// TIA Portal V17 export
// export: Created 2023-02-14T02:49:13.2032669Z, ExportSetting WithDefaults, DisplayName Totally Integrated Automation Portal, DisplayVersion V17, DisplayName TIA Portal Openness, DisplayVersion V17, DisplayName TIA Portal Teamcenter Gateway, DisplayVersion V17, DisplayName TIA Portal Version Control Interface, DisplayVersion V17, DisplayName SINAMICS Startdrive Advanced, DisplayVersion V17, DisplayName SINAMICS Startdrive G130, G150, S120, S150, SINAMICS MV, S210, DisplayVersion V17, DisplayName SINAMICS Startdrive G110M, G120, G120C, G120D, G120P, G115D, DisplayVersion V17, DisplayName STEP 7 Professional, DisplayVersion V17, DisplayName STEP 7 Safety, DisplayVersion V17, DisplayName WinCC Professional, DisplayVersion V17
DATA_BLOCK "Mix_to_CIP"   // DB221
{ S7_Optimized_Access := 'FALSE' }
VERSION : 0.1
// stored: AutoNumber false, DBAccessibleFromOPCUA true, DBAccessibleFromWebserver true, IsOnlyStoredInLoadMemory false, IsWriteProtectedInAS false
   VAR
      HeartBeat : Bool := TRUE;
      CIP_Request : Struct
         Header : Struct
            Header_CIP_Request : Bool;
         END_STRUCT;
         "Chili Awetan" : Struct
            "T-02.00_CIP_Request" : Bool;
            "T-03.00_CIP_Request" : Bool;
            "T-04.00_CIP_Request" : Bool;
         END_STRUCT;
         Tomato : Struct
            "T-05.00_CIP_Request" : Bool;
         END_STRUCT;
         ChiliFresh : Struct
            "T-06.00_CIP_Request" : Bool;
            "T-07.00_CIP_Request" : Bool;
            "T-08.00_CIP_Request" : Bool;
         END_STRUCT;
         Garlic : Struct
            "T-09.00_CIP_Request" : Bool;
         END_STRUCT;
         Vinegar : Struct
            "T-10.00_CIP_Request" : Bool;
         END_STRUCT;
         Homomixer : Struct
            "T-12.00_CIP_Tank_Request" : Bool;
            "T-12.00_CIP_LineToBlend_Request" : Bool;
            "T-13.00_CIP_Tank_Request" : Bool;
            "T-13.00_CIP_LineToBlend_Request" : Bool;
            "T-14.00_CIP_Tank_Request" : Bool;
            "T-14.00_CIP_LineToBlend_Request" : Bool;
         END_STRUCT;
         "Blending Cluster 1" : Struct
            "T-20.00_CIP_Request" : Bool;
            "T-21.00_CIP_Request" : Bool;
            "T-30.00_CIP_Request" : Bool;
            Blending_Cluster1_LineProduct_Request : Bool;
            Free_CIP_Req_1 : Bool;
            Free_CIP_Req_2 : Bool;
         END_STRUCT;
         "Blending Cluster 2" : Struct
            "T-31.00_CIP_Request" : Bool;
            "T-40.00_CIP_Request" : Bool;
            "T-41.00_CIP_Request" : Bool;
            Blending_Cluster2_LineProduct_Request : Bool;
            Free_CIP_Req_1 : Bool;
            Free_CIP_Req_2 : Bool;
         END_STRUCT;
         "Rework Cluster 1" : Struct
            "T-22.00_CIP_Request" : Bool;
         END_STRUCT;
         "Rework Cluster 2" : Struct
            "T-32.00_CIP_Request" : Bool;
         END_STRUCT;
         "Buffer Cluster 1" : Struct
            "T-61.00_CIP_Request" : Bool;
            "T-62.00_CIP_Request" : Bool;
            "T61&T62_CIP_LineToPasteur_Request" : Bool;
            "T-63.00_CIP_Request" : Bool;
            "T-64.00_CIP_Request" : Bool;
            "T63&T64_CIP_LineToPasteur_Request" : Bool;
         END_STRUCT;
         "Buffer Cluster 2" : Struct
            "T-65.00_CIP_Request" : Bool;
            "T-66.00_CIP_Request" : Bool;
            "T65&T66_CIP_LineToPasteur_Request" : Bool;
            "T-67.00_CIP_Request" : Bool;
            "T-68.00_CIP_Request" : Bool;
            "T67&T68_CIP_LineToPasteur_Request" : Bool;
         END_STRUCT;
         "Storage THE 4" : Struct
            "T-23.00_CIP_Tank_Request" : Bool;
            "T-23.00_CIP_Line_Request" : Bool;
            "T-24.00_CIP_Tank_Request" : Bool;
            "T-24.00_CIP_Line_Request" : Bool;
            THE4_LineProduct_CIP_Request : Bool;
         END_STRUCT;
         "Storage THE 5" : Struct
            "T-33.00_CIP_Tank_Request" : Bool;
            "T-34.00_CIP_Tank_Request" : Bool;
            "T33&T34_CIP_Line_Request" : Bool;
            "T-35.00_CIP_Tank_Request" : Bool;
            "T-35.00_CIP_Line_Request" : Bool;
            THE5_LineProduct_CIP_Request : Bool;
         END_STRUCT;
         "T-79.00_CIP_Tank_Request" : Bool;
         "T-79.00_CIP_Line_Request" : Bool;
         "T-81.00_CIP_Request" : Bool;
         "T-84.00_CIP_Request" : Bool;
         "T-85.00_CIP_Request" : Bool;
         Free_CIP_Req_6 : Bool;
         Free_CIP_Req_7 : Bool;
         Free_CIP_Req_8 : Bool;
         Free_CIP_Req_9 : Bool;
         Free_CIP_Req_10 : Bool;
         Free_CIP_Req_11 : Bool;
         Free_CIP_Req_12 : Bool;
         Free_CIP_Req_13 : Bool;
         Free_CIP_Req_14 : Bool;
         Free_CIP_Req_15 : Bool;
         Free_CIP_Req_16 : Bool;
         Osa_CIP_Req : Bool;
         Free_CIP_Req_18 : Bool;
         Free_CIP_Req_19 : Bool;
         Free_CIP_Req_20 : Bool;
         Free_CIP_Req_21 : Bool;
         Free_CIP_Req_22 : Bool;
         Free_CIP_Req_23 : Bool;
         Free_CIP_Req_24 : Bool;
      END_STRUCT;
      CIP_Line_OK : Struct
         Header : Struct
            Header_CIP_LineOK : Bool;
         END_STRUCT;
         "Chili Awetan" : Struct
            "T-02.00_CIP_LineOK" : Bool;
            "T-03.00_CIP_LineOK" : Bool;
            "T-04.00_CIP_LineOK" : Bool;
         END_STRUCT;
         Tomato : Struct
            "T-05.00_CIP_LineOK" : Bool;
         END_STRUCT;
         ChiliFresh : Struct
            "T-06.00_CIP_LineOK" : Bool;
            "T-07.00_CIP_LineOK" : Bool;
            "T-08.00_CIP_LineOK" : Bool;
         END_STRUCT;
         Garlic : Struct
            "T-09.00_CIP_LineOK" : Bool;
         END_STRUCT;
         Vinegar : Struct
            "T-10.00_CIP_LineOK" : Bool;
         END_STRUCT;
         Homomixer : Struct
            "T-12.00_CIP_LineOK" : Bool;
            "T-13.00_CIP_LineOK" : Bool;
            "T-14.00_CIP_LineOK" : Bool;
         END_STRUCT;
         "Blending Cluster 1" : Struct
            "T-20.00_CIP_LineOK" : Bool;
            "T-21.00_CIP_LineOK" : Bool;
            "T-30.00_CIP_LineOK" : Bool;
            Blending_Cluster1_LineProduct_LineOK : Bool;
            Free_CIP_LineOK_1 : Bool;
            Free_CIP_LineOK_2 : Bool;
         END_STRUCT;
         "Blending Cluster 2" : Struct
            "T-31.00_CIP_LineOK" : Bool;
            "T-40.00_CIP_LineOK" : Bool;
            "T-41.00_CIP_LineOK" : Bool;
            Blending_Cluster2_LineProduct_LineOK : Bool;
            Free_CIP_LineOK_1 : Bool;
            Free_CIP_LineOK_2 : Bool;
         END_STRUCT;
         "Rework Cluster 1" : Struct
            "T-22.00_CIP_LineOK" : Bool;
         END_STRUCT;
         "Rework Cluster 2" : Struct
            "T-32.00_CIP_LineOK" : Bool;
         END_STRUCT;
         "Buffer Cluster 1" : Struct
            "T-61.00_CIP_LineOK" : Bool;
            "T-62.00_CIP_LineOK" : Bool;
            "T61&T62_CIP_LineToPasteur_LineOK" : Bool;
            "T-63.00_CIP_LineOK" : Bool;
            "T-64.00_CIP_LineOK" : Bool;
            "T63&T64_CIP_LineToPasteur_LineOK" : Bool;
         END_STRUCT;
         "Buffer Cluster 2" : Struct
            "T-65.00_CIP_LineOK" : Bool;
            "T-66.00_CIP_LineOK" : Bool;
            "T65&T66_CIP_LineToPasteur_LineOK" : Bool;
            "T-67.00_CIP_LineOK" : Bool;
            "T-68.00_CIP_LineOK" : Bool;
            "T67&T68_CIP_LineToPasteur_LineOK" : Bool;
         END_STRUCT;
         "Storage THE 4" : Struct
            "T-23.00_CIP_LineOK" : Bool;
            "T-24.00_CIP_LineOK" : Bool;
            THE4_LineProduct_CIP_LineOK : Bool;
         END_STRUCT;
         "Storage THE 5" : Struct
            "T-33.00_CIP_Tank_LineOK" : Bool;
            "T-34.00_CIP_Tank_LineOK" : Bool;
            "T33&T34_CIP_Line_LineOK" : Bool;
            "T-35.00_CIP_Tank_LineOK" : Bool;
            THE5_LineProduct_CIP_LineOK : Bool;
         END_STRUCT;
         "T-79.00_CIP_LineOK" : Bool;
         "T-81.00_CIP_LineOK" : Bool;
         "T-84.00_CIP_LineOK" : Bool;
         "T-85.00_CIP_LineOK" : Bool;
         Free_CIP_LineOK_5 : Bool;
         Free_CIP_LineOK_6 : Bool;
         Free_CIP_LineOK_7 : Bool;
         Free_CIP_LineOK_8 : Bool;
         Free_CIP_LineOK_9 : Bool;
         Free_CIP_LineOK_10 : Bool;
         Free_CIP_LineOK_11 : Bool;
         Free_CIP_LineOK_12 : Bool;
         Free_CIP_LineOK_13 : Bool;
         Free_CIP_LineOK_14 : Bool;
         Free_CIP_LineOK_15 : Bool;
         Free_CIP_LineOK_16 : Bool;
         Osa_CIP_LineOK : Bool;
         Free_CIP_LineOK_18 : Bool;
         Free_CIP_LineOK_19 : Bool;
         Free_CIP_LineOK_20 : Bool;
         Free_CIP_LineOK_21 : Bool;
         Free_CIP_LineOK_22 : Bool;
         Free_CIP_LineOK_23 : Bool;
         Free_CIP_LineOK_24 : Bool;
      END_STRUCT;
   END_VAR
BEGIN
END_DATA_BLOCK
